(* PLC project PlcMain, Beckhoff Automation GmbH TwinCAT PLC Control 3.5.13.21 *)
(* stored: creationDateTime 2022-08-19T12:34:20.2352279, modificationDateTime 2022-08-19T12:34:20.2352279 *)

{attribute 'qualified_only'}
{attribute 'strict'}
TYPE State :
(
	Off,
	Busy,
	Ready,
	Done,
	Error,
	Setup
);
END_TYPE
